(* IEC 61131-3 sources: AXOpen/src/components.dukane.welders/ctrl/src/AxoIQSeriesWelder (part 3) *)

            _dword              :=  TO_DWORD(Outputs.OTF_Amp_Setpoint);
            _data_out[4]        :=  _dword.%B3;
            _data_out[5]        :=  _dword.%B2;
            _data_out[6]        :=  _dword.%B1;
            _data_out[7]        :=  _dword.%B0;

            _dword              :=  TO_DWORD(Outputs.ActiveSetupSelection);
            _data_out[8]        :=  _dword.%B3;
            _data_out[9]        :=  _dword.%B2;
            _data_out[10]       :=  _dword.%B1;
            _data_out[11]       :=  _dword.%B0;

            _dword              :=  TO_DWORD(Outputs.RunningSetupSelection);
            _data_out[12]       :=  _dword.%B3;
            _data_out[13]       :=  _dword.%B2;
            _data_out[14]       :=  _dword.%B1;
            _data_out[15]       :=  _dword.%B0;

            _dword              :=  TO_DWORD(Outputs.RunningMPCProbeSelection);
            _data_out[16]       :=  _dword.%B3;
            _data_out[17]       :=  _dword.%B2;
            _data_out[18]       :=  _dword.%B1;
            _data_out[19]       :=  _dword.%B0;

            _retval := WriteData(LADDR := TO_WORD(Config.HWIDs.HwID_PLC_to_iQ_Outputs),RECORD := _data_out);
            IF _retval > WORD#0 THEN
                Messenger.Activate(UINT#1231, eAxoMessageCategory#ProgrammingError);
                Status.Error.Id := UINT#1231;
                RETURN;
            END_IF;
        END_METHOD

        METHOD PUBLIC ClearError : IAxoTaskState
            ClearError := ClearErrorTask.Invoke(THIS);
        END_METHOD

        METHOD PUBLIC ChangeWeldingSetup : IAxoTaskState
            VAR_INPUT
                SetupNumber : UINT;
            END_VAR
            _setupNumber := SetupNumber;
            ChangeWeldingSetup := ChangeWeldingSetupTask.Invoke(THIS);
        END_METHOD

        METHOD PUBLIC ChangeWeldingProbe : IAxoTaskState
            VAR_INPUT
                ProbeNumber : UINT;
            END_VAR
            _probeNumber := ProbeNumber;
            ChangeWeldingProbe := ChangeWeldingProbeTask.Invoke(THIS);
        END_METHOD

        METHOD PUBLIC CycleStop : IAxoTaskState
            CycleStop := CycleStopTask.Invoke(THIS);
        END_METHOD

        METHOD PUBLIC RunWeldingWithTime : IAxoTaskState
            VAR_INPUT
                SetupNumber : UINT;
                ProbeNumber : UINT;
                WeldingTime : LTIME;
            END_VAR
            _setupNumber := SetupNumber;
            _probeNumber := ProbeNumber;
            _weldingTime := WeldingTime;
            RunWeldingWithTime := RunWeldingWithTimeTask.Invoke(THIS);
        END_METHOD

        METHOD PUBLIC TemplateMethod_10steps_6 : IAxoTaskState
            TemplateMethod_10steps_6 := TemplateTask_10steps_6.Invoke(THIS);
        END_METHOD

        METHOD PUBLIC TemplateMethod_20steps_1 : IAxoTaskState
            TemplateMethod_20steps_1 := TemplateTask_20steps_1.Invoke(THIS);
        END_METHOD

        METHOD PUBLIC TemplateMethod_20steps_2 : IAxoTaskState
            TemplateMethod_20steps_2 := TemplateTask_20steps_2.Invoke(THIS);
        END_METHOD

        METHOD PUBLIC TemplateMethod_20steps_3 : IAxoTaskState
            TemplateMethod_20steps_3 := TemplateTask_20steps_3.Invoke(THIS);
        END_METHOD

        METHOD PUBLIC TemplateMethod_20steps_4 : IAxoTaskState
            TemplateMethod_20steps_4 := TemplateTask_20steps_4.Invoke(THIS);
        END_METHOD

        METHOD PUBLIC TemplateMethod_20steps_5 : IAxoTaskState
            TemplateMethod_20steps_5 := TemplateTask_20steps_5.Invoke(THIS);
        END_METHOD

        METHOD PUBLIC TemplateMethod_20steps_6 : IAxoTaskState
            TemplateMethod_20steps_6 := TemplateTask_20steps_6.Invoke(THIS);
        END_METHOD

        METHOD PROTECTED OVERRIDE ManualControl
            _setupNumber := RequiredSetupNumber;
            _probeNumber := RequiredProbeNumber;
            _weldingTime := RequiredWeldingTime;
            THIS._isManuallyControllable := true;
        END_METHOD

        ///<summary>
        /// Restores this component into intial state.
        ///</summary>
        METHOD PUBLIC OVERRIDE Restore
            VAR
                _index : INT;
            END_VAR
            Status.Action.Id := UINT#0;
            Status.Error.Id  := UINT#0;

            _progress       :=   INT#0;
            _retVal    :=   WORD#0;

            FOR _index := 0 TO 19 DO
                _data_in[_index]    := BYTE#0;
                _data_out[_index]   := BYTE#0;
            END_FOR;

            FOR _index := 20 TO 139 DO
                _data_in[_index] := BYTE#0;
            END_FOR;

            _word           :=   WORD#0;
            _dword          :=   DWORD#0;

            _weldingTimer.OnDelay(THIS,FALSE,T#0S);

            ClearErrorTask.Restore();
            ChangeWeldingSetupTask.Restore();
            ChangeWeldingProbeTask.Restore();
            CycleStopTask.Restore();
            RunWeldingWithTimeTask.Restore();
            TemplateTask_10steps_6.Restore();
            TemplateTask_20steps_1.Restore();
            TemplateTask_20steps_2.Restore();
            TemplateTask_20steps_3.Restore();
            TemplateTask_20steps_4.Restore();
            TemplateTask_20steps_5.Restore();
            TemplateTask_20steps_6.Restore();
            HardwareDiagnosticsTask.Restore();

            Outputs.ClearSetup := FALSE;
            Outputs.RunScan := FALSE;
            Outputs.RunContinuously := FALSE;
            Outputs.RunWeld := FALSE;
            Outputs.RunTest := FALSE;
            Outputs.ClearError := FALSE;
            Outputs.OTF_AmplitudeEnable := FALSE;
            Outputs.CycleStop := FALSE;
            Outputs.FrontPanelLockout_0 := FALSE;
            Outputs.FrontPanelLockout_1 := FALSE;
            // Outputs.OTF_Amp_Setpoint := DINT#0;
            // Outputs.ActiveSetupSelection := DINT#0;
            // Outputs.RunningSetupSelection := DINT#0;
            // Outputs.RunningMPCProbeSelection := DINT#0;

            Status.Action.Id := UINT#50;
            RestoreTask.DoneWhen(TRUE);

        END_METHOD

        METHOD PRIVATE CallTimers
            VAR_INPUT
                signal : BOOL;
            END_VAR

            _infoTimer.OnDelay(THIS, signal AND Config.InfoTime > T#0S ,Config.InfoTime);
            _errorTimer.OnDelay(THIS, signal AND Config.ErrorTime > T#0S , Config.ErrorTime);

        END_METHOD

    END_CLASS
END_NAMESPACE

(* ---- Axo_IQ_SeriesWelder_Component_Status.st ---- *)
NAMESPACE AXOpen.Components.Dukane.Welders
    {S7.extern=ReadWrite}
    {#ix-attr:[Container(Layout.Stack)]}
    CLASS PUBLIC Axo_IQ_SeriesWelder_Component_Status EXTENDS AXOpen.Components.Abstractions.AxoComponent_Status
        VAR PUBLIC

        END_VAR
    END_CLASS
END_NAMESPACE

(* ---- Axo_IQ_SeriesWelder_CyclePartStatusBitDefinition.st ---- *)
NAMESPACE AXOpen.Components.Dukane.Welders
    {S7.extern=ReadWrite}
    {#ix-attr:[Container(Layout.Wrap)]}
    CLASS PUBLIC Axo_IQ_SeriesWelder_CyclePartStatusBitDefinition
        VAR PUBLIC
            {#ix-set:AttributeName = "<#LowerBadEnergyLimit#>"}
            LowerBadEnergyLimit : BOOL;
            {#ix-set:AttributeName = "<#LowerSuspectEnergyLimit#>"}
            LowerSuspectEnergyLimit : BOOL;
            {#ix-set:AttributeName = "<#UpperSuspectEnergyLimit#>"}
            UpperSuspectEnergyLimit : BOOL;
            {#ix-set:AttributeName = "<#UpperBadEnergyLimit#>"}
            UpperBadEnergyLimit : BOOL;
            // {#ix-set:AttributeName = "<#_4#>"}
            // _4 : BOOL;
            // {#ix-set:AttributeName = "<#_5#>"}
            // _5 : BOOL;
            // {#ix-set:AttributeName = "<#_6#>"}
            // _6 : BOOL;
            // {#ix-set:AttributeName = "<#_7#>"}
            // _7 : BOOL;
            {#ix-set:AttributeName = "<#LowerBadPowerLimit#>"}
            LowerBadPowerLimit : BOOL;
            {#ix-set:AttributeName = "<#LowerSuspectPowerLimit#>"}
            LowerSuspectPowerLimit : BOOL;
            {#ix-set:AttributeName = "<#UpperSuspectPowerLimit#>"}
            UpperSuspectPowerLimit : BOOL;
            {#ix-set:AttributeName = "<#UpperBadPowerLimit#>"}
            UpperBadPowerLimit : BOOL;
            // {#ix-set:AttributeName = "<#_12#>"}
            // _12 : BOOL;
            // {#ix-set:AttributeName = "<#_13#>"}
            // _13 : BOOL;
            // {#ix-set:AttributeName = "<#_14#>"}
            // _14 : BOOL;
            // {#ix-set:AttributeName = "<#_15#>"}
            // _15 : BOOL;
            {#ix-set:AttributeName = "<#LowerBadTimeLimit#>"}
            LowerBadTimeLimit : BOOL;
            {#ix-set:AttributeName = "<#LowerSuspectTimeLimit#>"}
            LowerSuspectTimeLimit : BOOL;
            {#ix-set:AttributeName = "<#UpperSuspectTimeLimit#>"}
            UpperSuspectTimeLimit : BOOL;
            {#ix-set:AttributeName = "<#UpperBadTimeLimit#>"}
            UpperBadTimeLimit : BOOL;
            // {#ix-set:AttributeName = "<#_20#>"}
            // _20 : BOOL;
            // {#ix-set:AttributeName = "<#_21#>"}
            // _21 : BOOL;
            // {#ix-set:AttributeName = "<#_22#>"}
            // _22 : BOOL;
            // {#ix-set:AttributeName = "<#_23#>"}
            // _23 : BOOL;
            {#ix-set:AttributeName = "<#GoodPart#>"}
            GoodPart : BOOL;
            {#ix-set:AttributeName = "<#BadPart#>"}
            BadPart : BOOL;
            {#ix-set:AttributeName = "<#SuspectPart#>"}
            SuspectPart : BOOL;
            // {#ix-set:AttributeName = "<#_27#>"}
            // _27 : BOOL;
            // {#ix-set:AttributeName = "<#_28#>"}
            // _28 : BOOL;
            // {#ix-set:AttributeName = "<#_29#>"}
            // _29 : BOOL;
            // {#ix-set:AttributeName = "<#_30#>"}
            // _30 : BOOL;
            // {#ix-set:AttributeName = "<#_31#>"}
            // _31 : BOOL;
        END_VAR
    END_CLASS
END_NAMESPACE

(* ---- Axo_IQ_SeriesWelder_PressPartStatusBitDefinition.st ---- *)
NAMESPACE AXOpen.Components.Dukane.Welders
    {S7.extern=ReadWrite}
    {#ix-attr:[Container(Layout.Wrap)]}
    CLASS PUBLIC Axo_IQ_SeriesWelder_PressPartStatusBitDefinition
        VAR PUBLIC
            {#ix-set:AttributeName = "<#Weld1Position#>"}
            Weld1Position : BOOL;
            {#ix-set:AttributeName = "<#ErrorStatus#>"}
            ErrorStatus : BOOL;
            // {#ix-set:AttributeName = "<#_26#>"}
            // _26 : BOOL;
            // {#ix-set:AttributeName = "<#_27#>"}
            // _27 : BOOL;
            // {#ix-set:AttributeName = "<#_28#>"}
            // _28 : BOOL;
            // {#ix-set:AttributeName = "<#_29#>"}
            // _29 : BOOL;
            // {#ix-set:AttributeName = "<#_30#>"}
            // _30 : BOOL;
            // {#ix-set:AttributeName = "<#_31#>"}
            // _31 : BOOL;
            {#ix-set:AttributeName = "<#TotalWeldTime#>"}
            TotalWeldTime : BOOL;
            {#ix-set:AttributeName = "<#TotalWeldDistance#>"}
            TotalWeldDistance : BOOL;
            {#ix-set:AttributeName = "<#TotalWeldEnergy#>"}
            TotalWeldEnergy : BOOL;
            {#ix-set:AttributeName = "<#HoldTime#>"}
            HoldTime: BOOL;
            {#ix-set:AttributeName = "<#HoldDistance#>"}
            HoldDistance: BOOL;
            {#ix-set:AttributeName = "<#TotalCycleTime#>"}
            TotalCycleTime : BOOL;
            {#ix-set:AttributeName = "<#FinalHoldPosition#>"}
            FinalHoldPosition : BOOL;
            {#ix-set:AttributeName = "<#Weld1PeakForce#>"}
            Weld1PeakForce : BOOL;
            {#ix-set:AttributeName = "<#Weld1Distance#>"}
            Weld1Distance : BOOL;
            {#ix-set:AttributeName = "<#Weld1Energy#>"}
            Weld1Energy : BOOL;
            {#ix-set:AttributeName = "<#Weld1Power#>"}
            Weld1Power : BOOL;
            {#ix-set:AttributeName = "<#Weld2Time#>"}
            Weld2Time : BOOL;
            {#ix-set:AttributeName = "<#Weld2Distance#>"}
            Weld2Distance : BOOL;
            {#ix-set:AttributeName = "<#Weld2Energy#>"}
            Weld2Energy : BOOL;
            {#ix-set:AttributeName = "<#Weld2Power#>"}
            Weld2Power : BOOL;
            {#ix-set:AttributeName = "<#Weld2Position#>"}
            Weld2Position : BOOL;
            {#ix-set:AttributeName = "<#TriggerTime#>"}
            TriggerTime : BOOL;
            {#ix-set:AttributeName = "<#TriggerPosition#>"}
            TriggerPosition : BOOL;
            {#ix-set:AttributeName = "<#AverageSensingVelocity#>"}
            AverageSensingVelocity : BOOL;
            {#ix-set:AttributeName = "<#TriggerPressure#>"}
            TriggerPressure : BOOL;
            {#ix-set:AttributeName = "<#TriggerForce#>"}
            TriggerForce : BOOL;
            {#ix-set:AttributeName = "<#TriggerDelayTime#>"}
            TriggerDelayTime : BOOL;
            {#ix-set:AttributeName = "<#TriggerDelayDistance#>"}
            TriggerDelayDistance : BOOL;
            {#ix-set:AttributeName = "<#Weld1Time#>"}
            Weld1Time : BOOL;
        END_VAR
    END_CLASS
END_NAMESPACE

(* ---- Axo_IQ_SeriesWelder_SystemInputs.st ---- *)
NAMESPACE AXOpen.Components.Dukane.Welders
    {S7.extern=ReadWrite}
    {#ix-attr:[Container(Layout.Wrap)]}
    CLASS PUBLIC Axo_IQ_SeriesWelder_SystemInputs
        VAR PUBLIC
            {#ix-set:AttributeName = "<#SystemErrorStatus#>"}
            SystemErrorStatus : Axo_IQ_SeriesWelder_ErrorStatusBitDefinition;
            {#ix-set:AttributeName = "<#SystemInitiateError#>"}
            SystemInitiateError : DInt;
            {#ix-set:AttributeName = "<#SystemProcessError#>"}
            SystemProcessError : Axo_IQ_SeriesWelder_ProcessErrorStatus;
            {#ix-set:AttributeName = "<#GeneratorState#>"}
            GeneratorState : DInt;
            {#ix-set:AttributeName = "<#RealTimeAmplitude#>"}
            RealTimeAmplitude : DInt;   // The current amplitude of the stack in units percent amplitude.
            {#ix-set:AttributeName = "<#RealTimeFrequency#>"}
            RealTimeFrequency : DInt;   // The current frequency of the stack in units of Hz.
            {#ix-set:AttributeName = "<#RealTimePower#>"}
            RealTimePower : DInt;   // The current driven power of the stack in units of Watts
            {#ix-set:AttributeName = "<#SystemStatus#>"}
            SystemStatus : Axo_IQ_SeriesWelder_SystemStatusBitDefinition;
            {#ix-set:AttributeName = "<#Temperature#>"}
            Temperature : DInt;   // The current internal temperature of the iQ in units of Degrees Celcius
            {#ix-set:AttributeName = "<#CycleCount#>"}
            CycleCount : DInt;   // Count of total number of cycles since power up (not influenced by a test cycle)
            {#ix-set:AttributeName = "<#GoodPartCount#>"}
            GoodPartCount : DInt;   // Count of total number of "good parts" as determined by the Process Limits.
            {#ix-set:AttributeName = "<#BadPartCount#>"}
            BadPartCount : DInt;   // Count of total number of "bad parts" as determined by the Process Limits.
            {#ix-set:AttributeName = "<#SuspectPartCount#>"}
            SuspectPartCount : DInt;   // Count of total number of "suspect parts" as determined by the Process Limits.
            {#ix-set:AttributeName = "<#AbortedPartCount#>"}
            AbortedPartCount : DInt;   // Count of total number of weld cycles that failed to trigger since power up (not
            {#ix-set:AttributeName = "<#CyclePartStatus#>"}
            CyclePartStatus : Axo_IQ_SeriesWelder_CyclePartStatusBitDefinition;
            {#ix-set:AttributeName = "<#CycleWeldTime#>"}
            CycleWeldTime : DInt;   // Total Weld Time of the last cycle, units of mS .
            {#ix-set:AttributeName = "<#CycleWeldPeakPower#>"}
            CycleWeldPeakPower : DInt;   // Peak Weld Power of last cycle, units of Watts .
            {#ix-set:AttributeName = "<#CycleWeldEnergy#>"}
            CycleWeldEnergy : DInt;   // Total Weld Energy of last cycle, units of Joules .
            {#ix-set:AttributeName = "<#ActiveSetup#>"}
            ActiveSetup : DInt;   // Weld process control "setup" that the PLC access,values range from 1 to 16.
            {#ix-set:AttributeName = "<#RunningSetup#>"}
            RunningSetup : DInt;   // Commands the weld process control setup that the iQ will use on the next cycle,
            {#ix-set:AttributeName = "<#RunningMPCProbe#>"}
            RunningMPCProbe : DInt;   // Commands the MPC probe selection that the iQ will use on the next cycle, values
            {#ix-set:AttributeName = "<#SelectedInputVoltage#>"}
            SelectedInputVoltage : DInt;
            {#ix-set:AttributeName = "<#RealTimePosition#>"}
            RealTimePosition : DInt;
            {#ix-set:AttributeName = "<#RealTimeVelocity#>"}
            RealTimeVelocity : DInt;
            {#ix-set:AttributeName = "<#PressPartStatus_Bad_lo#>"}
            PressPartStatus_Bad_lo : Axo_IQ_SeriesWelder_PressPartStatusBitDefinition;
            {#ix-set:AttributeName = "<#PressPartStatus_Sus_lo#>"}
            PressPartStatus_Sus_lo : Axo_IQ_SeriesWelder_PressPartStatusBitDefinition;
            {#ix-set:AttributeName = "<#PressPartStatus_Sus_hi#>"}
            PressPartStatus_Sus_hi : Axo_IQ_SeriesWelder_PressPartStatusBitDefinition;
            {#ix-set:AttributeName = "<#PressPartStatus_Bad_hi#>"}
            PressPartStatus_Bad_hi : Axo_IQ_SeriesWelder_PressPartStatusBitDefinition;
            {#ix-set:AttributeName = "<#CycleTriggerTime#>"}
            CycleTriggerTime : DInt;
            {#ix-set:AttributeName = "<#CycleTriggerPosition#>"}
            CycleTriggerPosition : DInt;
            {#ix-set:AttributeName = "<#CycleTriggerDelayTime#>"}
            CycleTriggerDelayTime : DInt;
            {#ix-set:AttributeName = "<#CycleTriggerDelayDistance#>"}
            CycleTriggerDelayDistance : DInt;
            {#ix-set:AttributeName = "<#CycleWeld1Distance#>"}
            CycleWeld1Distance : DInt;
            {#ix-set:AttributeName = "<#CycleWeld1Position#>"}
            CycleWeld1Position : DInt;
            {#ix-set:AttributeName = "<#CycleTotalTime#>"}
            CycleTotalTime : DInt;
        END_VAR
    END_CLASS
END_NAMESPACE

(* ---- Axo_IQ_SeriesWelder_SystemStatusBitDefinition.st ---- *)
NAMESPACE AXOpen.Components.Dukane.Welders
    {S7.extern=ReadWrite}
    {#ix-attr:[Container(Layout.Wrap)]}
    CLASS PUBLIC Axo_IQ_SeriesWelder_SystemStatusBitDefinition
        VAR PUBLIC
            // {#ix-set:AttributeName = "<#res_bit24#>"}
            // res_bit24 : BOOL;   // bit24
            // {#ix-set:AttributeName = "<#res_bit25#>"}
            // res_bit25 : BOOL;   // bit25
            // {#ix-set:AttributeName = "<#res_bit26#>"}
            // res_bit26 : BOOL;   // bit26
            // {#ix-set:AttributeName = "<#res_bit27#>"}
            // res_bit27 : BOOL;   // bit27
            // {#ix-set:AttributeName = "<#res_bit28#>"}
            // res_bit28 : BOOL;   // bit28
            // {#ix-set:AttributeName = "<#res_bit29#>"}
            // res_bit29 : BOOL;   // bit29
            // {#ix-set:AttributeName = "<#res_bit30#>"}
            // res_bit30 : BOOL;   // bit30
            {#ix-set:AttributeName = "<#SetupChanged#>"}
            SetupChanged : BOOL;   // bit31
            {#ix-set:AttributeName = "<#InCycle#>"}
            InCycle : BOOL;   // bit16
            {#ix-set:AttributeName = "<#InCycle_No_AB#>"}
            InCycle_No_AB : BOOL;   // bit17
            {#ix-set:AttributeName = "<#OverTemp#>"}
            OverTemp : BOOL;   // bit18
            {#ix-set:AttributeName = "<#In_AfterBurst#>"}
            In_AfterBurst : BOOL;   // bit19
            {#ix-set:AttributeName = "<#In_Test#>"}
            In_Test : BOOL;   // bit20
            {#ix-set:AttributeName = "<#In_TestScan#>"}
            In_TestScan : BOOL;   // bit21
            {#ix-set:AttributeName = "<#MPC_Present#>"}
            MPC_Present : BOOL;   // bit22
            // {#ix-set:AttributeName = "<#res_bit23#>"}
            // res_bit23 : BOOL;   // bit23
            {#ix-set:AttributeName = "<#PowerOK#>"}
            PowerOK : BOOL;   // bit8
            {#ix-set:AttributeName = "<#MPC_Ready#>"}
            MPC_Ready : BOOL;   // bit9
            {#ix-set:AttributeName = "<#Ready#>"}
            Ready : BOOL;   // bit10
            {#ix-set:AttributeName = "<#Any_Fault#>"}
            Any_Fault : BOOL;   // bit11
            {#ix-set:AttributeName = "<#Overload#>"}
            Overload : BOOL;   // bit12
            {#ix-set:AttributeName = "<#Estop#>"}
            Estop : BOOL;   // bit13
            {#ix-set:AttributeName = "<#Online#>"}
            Online : BOOL;   // bit14
            {#ix-set:AttributeName = "<#In_Hold#>"}
            In_Hold : BOOL;   // bit15
            {#ix-set:AttributeName = "<#Good_Part#>"}
            Good_Part : BOOL;   // bit0
            {#ix-set:AttributeName = "<#Bad_Part#>"}
            Bad_Part : BOOL;   // bit1
            {#ix-set:AttributeName = "<#Suspect_Part#>"}
            Suspect_Part : BOOL;   // bit2
            {#ix-set:AttributeName = "<#CycleStartReject#>"}
            CycleStartReject : BOOL;   // bit3
            {#ix-set:AttributeName = "<#Amplitude_Regulation#>"}
            Amplitude_Regulation : BOOL;   // bit4
            {#ix-set:AttributeName = "<#Power_Regulation#>"}
            Power_Regulation : BOOL;   // bit5
            {#ix-set:AttributeName = "<#Trigger_Status#>"}
            Trigger_Status : BOOL;   // bit6
            {#ix-set:AttributeName = "<#US_Status#>"}
            US_Status : BOOL;   // bit7
        END_VAR
    END_CLASS
END_NAMESPACE
